Staubli VAL3: countBool2D.pgx

public program countBool2D(bool& x_bInput[] (dimensions=2), num& x_nResult)
  local num l_nElement
  local num l_nDim[2]
begin

  x_nResult = 0

  for l_nDim[0] = 0 to size(x_bInput,1)-1
    for l_nDim[1] = 0 to size(x_bInput,2)-1
        if x_bInput[l_nDim[0], l_nDim[1]] == true
          x_nResult = x_nResult+1
        endIf
    endFor
  endFor

end
